TYPE RedundancyParameters :
STRUCT
END_STRUCT
END_TYPE

(* stored: Version 1.1.0.1, ProductVersion 3.1.4024.6
   DUT RedundancyParameters: Id {88fa84a7-ca29-4a9f-886b-67649cb7b6a3} *)
